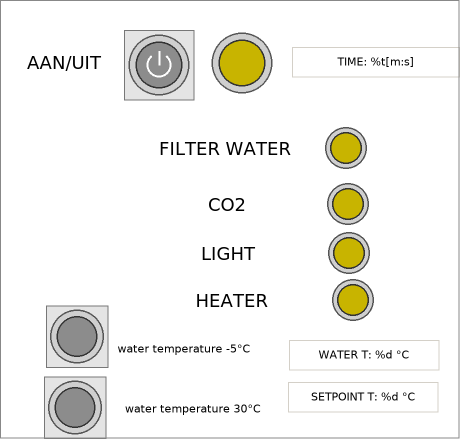
VISUALIZATION Visualization  // 460x439
    Lamp1 (207,28 70x70), variable: GVL.ix_START, style: Lamp-Lamp1-Yellow
    PowerSwitch (124,30 70x70), variable: GVL.ix_START, behaviour: TOGGLE, style: Switch-PowerSwitch-Gray
    Label (14,48 101x30), "AAN/UIT"
    Lamp1 (322,124 48x48), variable: GVL.ox_FILTER_WATER, style: Lamp-Lamp1-Yellow
    Textfield (288,382 150x30), "SETPOINT T: %d °C", text variable: GVL.id_TEMP_SETPOINT
    PushSwitch (46,305 62x63), variable: GVL.ix_COOLDOWN, behaviour: TOGGLE, style: Switch-PushSwitch-Gray
    Label (109,334 150x30), "water temperature -5°C"
    Label (138,134 174x30), "FILTER WATER"
    Lamp1 (324,180 48x48), variable: GVL.ox_CO2, style: Lamp-Lamp1-Yellow
    Label (140,190 174x30), "CO2"
    Lamp1 (325,229 48x48), variable: GVL.ox_LIGHT, style: Lamp-Lamp1-Yellow
    Label (141,239 174x30), "LIGHT"
    Lamp1 (329,276 48x48), variable: GVL.ox_HEATER, style: Lamp-Lamp1-Yellow
    Label (145,286 174x30), "HEATER"
    PushSwitch (44,376 62x63), variable: GVL.ix_TEMPRESET, behaviour: TOGGLE, style: Switch-PushSwitch-Gray
    Label (118,394 150x30), "water temperature 30°C"
    Textfield (292,47 168x30), "TIME: %t[m:s]", text variable: MAIN.FilterCycle1.T_CYCLE.ET
    Textfield (289,340 150x30), "WATER T: %d °C", text variable: GVL.id_TEMP_SENSOR
END_VISUALIZATION

(* stored: Version 1.1.0.1, ProductVersion 3.1.4024.15
   Visu Visualization: Id {cd8d33d6-dd8c-4cca-b370-5e78cd1dcb15} *)
